FUNCTION_BLOCK Q_ChildPosition_AI (* Command change child position ( Part 6 - F.16 ) — X/Y position via AI adapter sockets (wraps Q_ChildPosition) *)
  (* Standard: ISO 11783-6; Description: Copyright (c) 2026 Meisterschulen am Ostbahnhof This program and the accompanying materials are made available under the terms of the Eclipse Public License 2.0 which is available at https://www.eclipse.org/legal/epl-2.0/ SPDX-License-Identifier: EPL-2.0 AI adapter wrapper around Q_ChildPosition: s16Xposition and s16Yposition are each received via their own AI adapter socket instead of a plain REQ/data pair. Either socket's own event triggers a position update (Q_ChildPosition.REQ), reading whichever INT value currently sits on both sockets' D1. Object IDs (u16ObjId/u16ObjIdParent) are unchanged plain INIT inputs, same as Q_ChildPosition itself. *)
  (* Version 1.1, 2026-09-05, Franz Höpfinger, Meisterschulen am Ostbahnhof, Add xScale flag *)
  (* Version 1.0, 2026-09-05, Franz Höpfinger, Meisterschulen am Ostbahnhof, initial API and implementation and/or initial documentation *)
  PACKAGE isobus::UT::Q;
  IMPORT isobus::UT::Q::Q_ChildPosition;
  IMPORT isobus::UT::Q::const::IDs::ID_NULL;
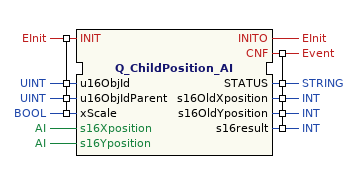
  EVENT_INPUT
    INIT : EInit WITH u16ObjId, u16ObjIdParent, xScale; (* Service Initialization *)
  END_EVENT
  EVENT_OUTPUT
    INITO : EInit; (* Initialization Confirm *)
    CNF WITH STATUS, s16OldXposition, s16OldYposition, s16result; (* Confirmation of Requested Service *)
  END_EVENT
  VAR_INPUT
    u16ObjId : UINT := ID_NULL; (* Object ID *)
    u16ObjIdParent : UINT := ID_NULL; (* Parent object ID *)
    xScale : BOOL := FALSE; (* FALSE (default) = bypass, send s16Xposition/s16Yposition through unchanged. TRUE = scale them by the DM/SKM factor for u16ObjIdParent. *)
  END_VAR
  VAR_OUTPUT
    STATUS : STRING; (* Service Status - passthrough from the internal Q_ChildPosition *)
    s16OldXposition : INT; (* Old X position - passthrough from the internal Q_ChildPosition *)
    s16OldYposition : INT; (* Old Y position - passthrough from the internal Q_ChildPosition *)
    s16result : INT; (* retval - passthrough from the internal Q_ChildPosition, see Q_ChildPosition *)
  END_VAR
  SOCKETS
    s16Xposition : adapter::types::unidirectional::AI; (* New X position relative to the top left corner of parent object *)
    s16Yposition : adapter::types::unidirectional::AI; (* New Y position relative to the top left corner of parent object *)
  END_SOCKETS
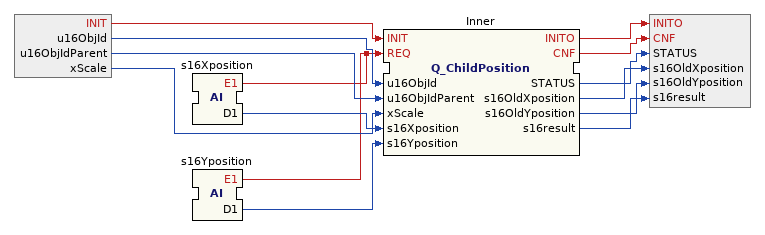
  FBS
    Inner : isobus::UT::Q::Q_ChildPosition;
  END_FBS
  EVENT_CONNECTIONS
    INIT TO Inner.INIT;
    s16Xposition.E1 TO Inner.REQ;
    s16Yposition.E1 TO Inner.REQ;
    Inner.INITO TO INITO;
    Inner.CNF TO CNF;
  END_CONNECTIONS
  DATA_CONNECTIONS
    u16ObjId TO Inner.u16ObjId;
    u16ObjIdParent TO Inner.u16ObjIdParent;
    xScale TO Inner.xScale;
    s16Xposition.D1 TO Inner.s16Xposition;
    s16Yposition.D1 TO Inner.s16Yposition;
    Inner.STATUS TO STATUS;
    Inner.s16OldXposition TO s16OldXposition;
    Inner.s16OldYposition TO s16OldYposition;
    Inner.s16result TO s16result;
  END_CONNECTIONS
END_FUNCTION_BLOCK
